FUNCTION_BLOCK Multicast_TwoCTL (* Composite Function Block Type *)
  (* Standard: 61499-2 *)
  (* Version 0.2, 2003-12-05, JHC, Rockwell Automation, Renamed from NEWCOMPFB. *)
  (* Version 0.1, 2002-01-08, JHC, Rockwell Automation, Added DLY FB as example. *)
  (* Version 0.0, 2000-05-27, JHC, Rockwell Automation *)
  (* Compiler header: package fb.rt.cs725; *)
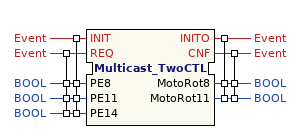
  EVENT_INPUT
    INIT WITH PE8, PE11, PE14; (* Initialization Request *)
    REQ WITH PE8, PE14, PE11; (* Normal Execution Request *)
  END_EVENT
  EVENT_OUTPUT
    INITO WITH MotoRot8, MotoRot11; (* Initialization Confirm *)
    CNF WITH MotoRot8, MotoRot11; (* Execution Confirmation *)
  END_EVENT
  VAR_INPUT
    PE8 : BOOL; (* Input event qualifier *)
    PE11 : BOOL;
    PE14 : BOOL;
  END_VAR
  VAR_OUTPUT
    MotoRot8 : BOOL; (* Output event qualifier *)
    MotoRot11 : BOOL;
  END_VAR
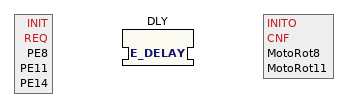
  FBS
    DLY : E_DELAY;
  END_FBS
END_FUNCTION_BLOCK
